PROGRAM Main4
VAR
END_VAR

END_PROGRAM

(* stored: Version 1.1.0.1, ProductVersion 3.1.4024.11
   POU Main4: Id {1f59f9a7-d9e9-4ba7-9582-5be5c950cb6a}, SpecialFunc None *)
